// TIA Portal V16 export
// export: Created 2023-03-29T11:05:03.7599548Z, ExportSetting WithDefaults, DisplayName Totally Integrated Automation Portal, DisplayVersion V16 Update 6, DisplayName TIA Portal Version Control Interface, DisplayVersion V16 Update 2, DisplayName TIA Portal Openness, DisplayVersion V16 Update 6, DisplayName STEP 7 Professional, DisplayVersion V16 Update 6, DisplayName STEP 7 Safety, DisplayVersion V16, DisplayName WinCC Advanced, DisplayVersion V16 Update 6
VAR_GLOBAL   // PLC tag table "P1"
   inputReadyP1 AT %M81.4 : Bool;   // sugnał gotowość / Gotowość napędu
   inputRunF_P1 AT %M81.5 : Bool;   // stycznik falownik / Potwierdzenie pracy z falownika
   inputRunS_P1 AT %M81.6 : Bool;   // stycznik softstart / Powierdzenie pracy z sieci
   CMD_inverter_P1 AT %M81.7 : Bool;   // Stycznik Falownik
   CMD_network_P1 AT %M82.0 : Bool;   // Stycznik Sieć
   setCMD_FP1 AT %M207.0 : Bool;   // Znacznik sterowania w trybie falownik dlaP1
   setCMD_SP1 AT %M207.1 : Bool;   // Znacznik sterowania w trybie sieć
   IsReady_P1 AT %M17.0 : Bool;   // Znacznik gotowości napędu
   Hour_Work_P1 AT %MD36 : DWord;   // Licznik pracy
   Set_HWork_P1 AT %M19.0 : Bool;   // Znacznik ustawienia aktywnej do pracy (po porównaniu liczników pracy)
   IsRunInverter_P1 AT %M211.3 : Bool;   // Potwierdzenie pracy z falownika
   IsRunNetwork_P1 AT %M217.0 : Bool;   // Potwierdzenie pracy z sieci
   Is_extras_K1_P1 AT %M218.4 : Bool;   // Znacznik motor dodatkowy nr 1
   setSUPV_FP1 AT %M12.0 : Bool;   // Znacznik polecenia startu z falownika
   IsRun_P1 AT %M10.4 : Bool;   // Potwierdzenie pracy
   setSUPV_SP1 AT %M12.7 : Bool;   // Znacznik polecenia startu z sieci
   "Ustaw alarm P1" AT %M1040.1 : Bool;   // symulacyjny bit alarmu
   CMD_soft_P1 AT %M84.7 : Bool;   // sygnał z softstart potwierdzenie pracy / sygnał on/off soft-start
   CB_CMD_P1 AT %M12.4 : Bool;   // Znacznik polecenia on/off przekaźnik napędu
   resetFault_SoftStart_P1 AT %M50.0 : Bool;   // sygnał resetu softstart
   bitH_Alarm_P1 AT %M22.0 : Bool;   // Alarm - kopia bitu z instancji statusu napędu
   bitH_REM_P1 AT %M22.2 : Bool;   // Zdalna - kopia bitu z instancji statusu napędu
   bitH_RUN_P1 AT %M22.3 : Bool;   // Praca - kopia bitu z instancji statusu napędu
   bitH_OFF_P1 AT %M22.4 : Bool;   // Polecenie OFF - kopia bitu z instancji statusu napędu
   bitH_ON_P1 AT %M22.5 : Bool;   // Polecenie ON - kopia bitu z instancji statusu napędu
   bitH_Res_P1 AT %M22.6 : Bool;   // Reset - kopia bitu z instancji statusu napędu
   bitH_Aut_Man_P1 AT %M22.7 : Bool;   // Aut=1 Man=0 - kopia bitu z instancji statusu napędu
   Is_extras_K3_P1 AT %M17.7 : Bool;   // Znacznik motor dodatkowy nr 3
   Is_extras_K2_P1 AT %M218.7 : Bool;   // Znacznik motor dodatkowy nr 2
   off_add_K1_P1 AT %M52.0 : Bool;   // sterowanie wyłączeniem selektywnym dodatkowej
   off_add_K2_P1 AT %M52.1 : Bool;   // sterowanie wyłączeniem selektywnym dodatkowej
   off_add_K3_P1 AT %M52.2 : Bool;   // sterowanie wyłączeniem selektywnym dodatkowej
   off_add_K4_P1 AT %M53.4 : Bool;   // sterowanie wyłączeniem selektywnym dodatkowej
   Set_50Hz_M AT %M217.6 : Bool;   // Znacznik pamięci podtrzymujący przełączenie na sieć
   Mem_Res_setCMD_MC_P1 AT %M223.0 : Bool;   // pamięć zbocza załączenia timera blokowania stycznika falowni
   CMD_ErrorSet_NetworkP1 AT %M221.3 : Bool;   // Znacznik sterowania awaryjnego pracą pompy bez falownika
END_VAR
